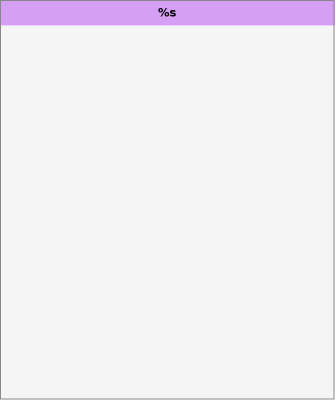
VISUALIZATION Uc_EntryDetail  // 335x400
    Rectangle (0,0 335x25), "%s", text variable: stVisu.sName
        OnMouseClick: write the text variable via Default
    Rectangle (0,26 335x373), text variable: stVisu.sName, colour variable: colCompBg
END_VISUALIZATION

(* stored: Version 1.1.0.1
   Visu Uc_EntryDetail: Id {4c339a8b-d561-462b-ae8c-e49b09f46e53} *)
